// TwinCAT 3 PLC project Untitled1
// ProgramVersion: 3.1.4024.0
// libraries:
//   Tc2_MC2, * (Beckhoff Automation GmbH)
//   Tc2_Standard, * (Beckhoff Automation GmbH)
//   Tc2_System, * (Beckhoff Automation GmbH)
//   Tc3_Module, * (Beckhoff Automation GmbH)
// project tree:
//   GVLs/ GVL.TcGVL
//   / PlcTask.TcTTO (not stored)
//   POUs/ MAIN.TcPOU
// real-time tasks:
//   TASK PlcTask: cycle T#10ms, priority 20, ADS port 350
// motion (NC):
//   TASK NC-Task 1 SAF: cycle T#2ms, priority 4, ADS port 501
//   TASK NC-Task 1 SVB: cycle T#10ms, priority 8, ADS port 511
//   AXIS Axis 1 (id 1)
//     Dynamic: AccelerationMaximum=150000, DecelerationMaximum=150000, Acceleration=5566, Deceleration=5566, Jerk=5566
//     Velo: SlowManual=5000, FastManual=150000, Maximum=150000
//     PositionAreaControl: Enable=false
//     TargetPosControl: Enable=false
//     OtherSettings: AllowMotionCmdToSlave=true
//     encoder EncType=19
//       EncPara: ScaleFactorNumerator=1, MaxCount=#xffffffff
//     drive DrvType=16
//       DrvPara: MaxCount=#xffffffff, DriveControlDWord=#x00020000
//         Analog: VeloReferenz=150000, TorqueSetpointScale=10, ScaleFactorActTorque=0.1
//         TimeComp: TaskDelayCycles=1
//     controller CtrType=1
//       CtrPara: PriorControlFactor=1
//         PosDiffControl: Enable=false
//         Observer: BandWidth=20
// I/O:
//   DEVICE Device 1 (EtherCAT), AmsNetId 192.168.1.160.2.1
//     Drive 1 (ZeroErr Driver) [ZeroErr Driver]
// variable links:
//   NC-Task 1 SAF/Axes/Axis 1 <-> Device 1 (EtherCAT)/Drive 1 (ZeroErr Driver)
//     Drive/Inputs/In/nDataIn1 <-> Transmit PDO mapping 0/Following error actual value
//     Drive/Inputs/In/nDataIn3[1] <-> Transmit PDO mapping 0/Torque Actual Value
//     Drive/Inputs/In/nDcOutputTime <-> InfoData/DcOutputShift
//     Drive/Inputs/In/nState1 <-> Transmit PDO mapping 0/Status word
//     Drive/Inputs/In/nState2 <-> Transmit PDO mapping 0/Status word @bit 8
//     Drive/Inputs/In/nState4 @bit 1 <-> WcState/InputToggle
//     Drive/Inputs/In/nState4 <-> WcState/WcState
//     Drive/Inputs/In/nState5 <-> Transmit PDO mapping 0/Modes of operation display
//     Drive/Outputs/Out/nCtrl1 <-> Receive PDO mapping 0/Control word
//     Drive/Outputs/Out/nCtrl2 <-> Receive PDO mapping 0/Control word @bit 8
//     Drive/Outputs/Out/nCtrl5 <-> Receive PDO mapping 0/Modes of operation
//     Drive/Outputs/Out/nDataOut1 <-> Receive PDO mapping 0/Target Position
//     Drive/Outputs/Out/nDataOut2 <-> Receive PDO mapping 0/Target Velocity
//     Drive/Outputs/Out/nDataOut3[1] <-> Receive PDO mapping 0/Torque Offset
//     Drive/Outputs/Out/nDataOut4[0] <-> Receive PDO mapping 0/Target Torque
//     Enc/Inputs/In/nDataIn1 <-> Transmit PDO mapping 0/Position actual value
//     Enc/Inputs/In/nDataIn7 <-> Transmit PDO mapping 0/Actual velocity
//     Enc/Inputs/In/nDcInputTime <-> InfoData/DcInputShift
//     Enc/Inputs/In/nState4 @bit 1 <-> WcState/InputToggle
//     Enc/Inputs/In/nState4 <-> WcState/WcState
//   Untitled1/Untitled1 Instance <-> NC-Task 1 SAF/Axes/Axis 1
//     PlcTask Inputs/MAIN.axis1.NcToPlc <-> Outputs/ToPlc
//     PlcTask Outputs/MAIN.axis1.PlcToNc <-> Inputs/FromPlc

// ---- GVLs/GVL.TcGVL
{attribute 'qualified_only'}
VAR_GLOBAL
	Actual_Velocity   AT%I*   :DINT  := 0;
	


	Control_word      AT%Q*   :UINT  := 0;
	int_val           AT%Q*   :INT   := 0;
	Target_Velocity   AT%Q*   :DINT  := 0;	
END_VAR

// ---- POUs/MAIN.TcPOU
PROGRAM MAIN
VAR
	BOOL1 :BOOL;
	axis1: AXIS_REF;
	
	fbPower: MC_Power;
    fbMoveAbsolute: MC_MoveAbsolute;
    fbMoveVelocity: MC_MoveVelocity;

    bEnable: BOOL := FALSE; (* 电机使能变量 *)
    bMove: BOOL := FALSE; (* 电机移动指令变量 *)
	
	fbJog: MC_Jog;  (* Jog 功能块 *)
 
    bJogForward: BOOL := FALSE;  (* 向前 Jog 的指令 *)
    bJogBackward: BOOL := FALSE; (* 向后 Jog 的指令 *)
    JogSpeed: LREAL := 500.0;    (* Jog 的速度 *)
	
	LRvelocity : LREAL  := 10000;
	
	fbTorqueControl: MC_TorqueControl;  (* 力矩控制功能块 *)

    bTorqueControl: BOOL := FALSE; (* 力控模式启动标志 *)
    TorqueValue: LREAL := 5.0;   (* 施加的力矩 *)
    MaxTorque: LREAL := 10.0;    (* 最大允许力矩 *)
    MinTorque: LREAL := -10.0;   (* 最小允许力矩 *)
    MaxVelocity: LREAL := 10000.0;    (* 最大允许速度 *)
    MinVelocity: LREAL := -10000.0;   (* 最小允许速度 *)
	
END_VAR


(* 电机使能 *)
fbPower(Axis := Axis1, Enable := bEnable, Enable_Positive := TRUE, Enable_Negative := TRUE);

(* 绝对位置移动 *)
fbMoveAbsolute(Axis := Axis1, Position := 0, Execute := bMove, Velocity := 50000.0, Acceleration := 1000.0, Deceleration := 1000.0, Jerk := 1000.0);

fbTorqueControl(Axis := Axis1, Torque := TorqueValue, Execute := bTorqueControl, TorqueRamp := 1000.0,VelocityLimitHigh := MaxVelocity, VelocityLimitLow := MinVelocity);

(* 前向 Jog 操作 *)
//fbJog(Axis := Axis1, JogForward := bJogForward, JogBackwards := bJogBackward, Velocity := JogSpeed, Acceleration := 1000.0, Deceleration := 1000.0, Jerk := 1000.0);

(* 如果需要速度控制，也可以使用 MC_MoveVelocity 函数 *)
//fbMoveVelocity(Axis := Axis1, Velocity := LRvelocity, Execute := bMove, Acceleration := 10000.0, Deceleration := 10000.0, Jerk := 1000.0);

END_PROGRAM
